TYPE ADSLoggerTestsystem :
STRUCT
  logging: EventRunner;
  event: Event := (logging:=logging);
  logger: ADSLogger := (disable_ads_output := TRUE);
END_STRUCT
END_TYPE

(* stored: Version 1.1.0.1, ProductVersion 3.1.4024.9
   DUT ADSLoggerTestsystem: Id {b1b05fc6-025d-4721-919d-ee911000e64d} *)
